FUNCTION_BLOCK RingToken (* Basic Function Block Type *)
  (* Standard: 61499-2 *)
  (* Version 0.2, 2003-12-04, JHC, Rockwell Automation, Renamed for better indexing. *)
  (* Version 0.1, 2002-11-05, JHC, Rockwell Automation, Corrected missing ST element in Algorithm REQ. *)
  (* Version 0.0, 2000-05-30, JHC, Rockwell Automation *)
  (* Compiler header: package fb.rt.cs725; *)
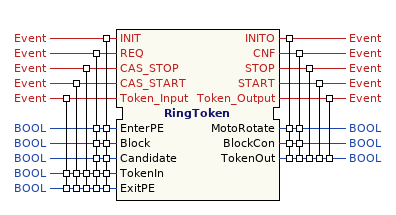
  EVENT_INPUT
    INIT WITH EnterPE, Block, Candidate, TokenIn, ExitPE; (* Initialization Request *)
    REQ WITH EnterPE, Block, Candidate, TokenIn, ExitPE; (* Normal Execution Request *)
    CAS_STOP WITH TokenIn, ExitPE;
    CAS_START WITH TokenIn, ExitPE;
    Token_Input WITH TokenIn, ExitPE;
  END_EVENT
  EVENT_OUTPUT
    INITO WITH MotoRotate, BlockCon, TokenOut; (* Initialization Confirm *)
    CNF WITH MotoRotate, BlockCon, TokenOut; (* Execution Confirmation *)
    STOP WITH TokenOut;
    START WITH TokenOut;
    Token_Output WITH TokenOut;
  END_EVENT
  VAR_INPUT
    EnterPE : BOOL; (* Input event qualifier *)
    Block : BOOL;
    Candidate : BOOL;
    TokenIn : BOOL;
    ExitPE : BOOL;
  END_VAR
  VAR_OUTPUT
    MotoRotate : BOOL; (* Output event qualifier *)
    BlockCon : BOOL;
    TokenOut : BOOL;
  END_VAR
  VAR
    lastPE : BOOL := 1;
    lastBlock : BOOL := 0;
  END_VAR
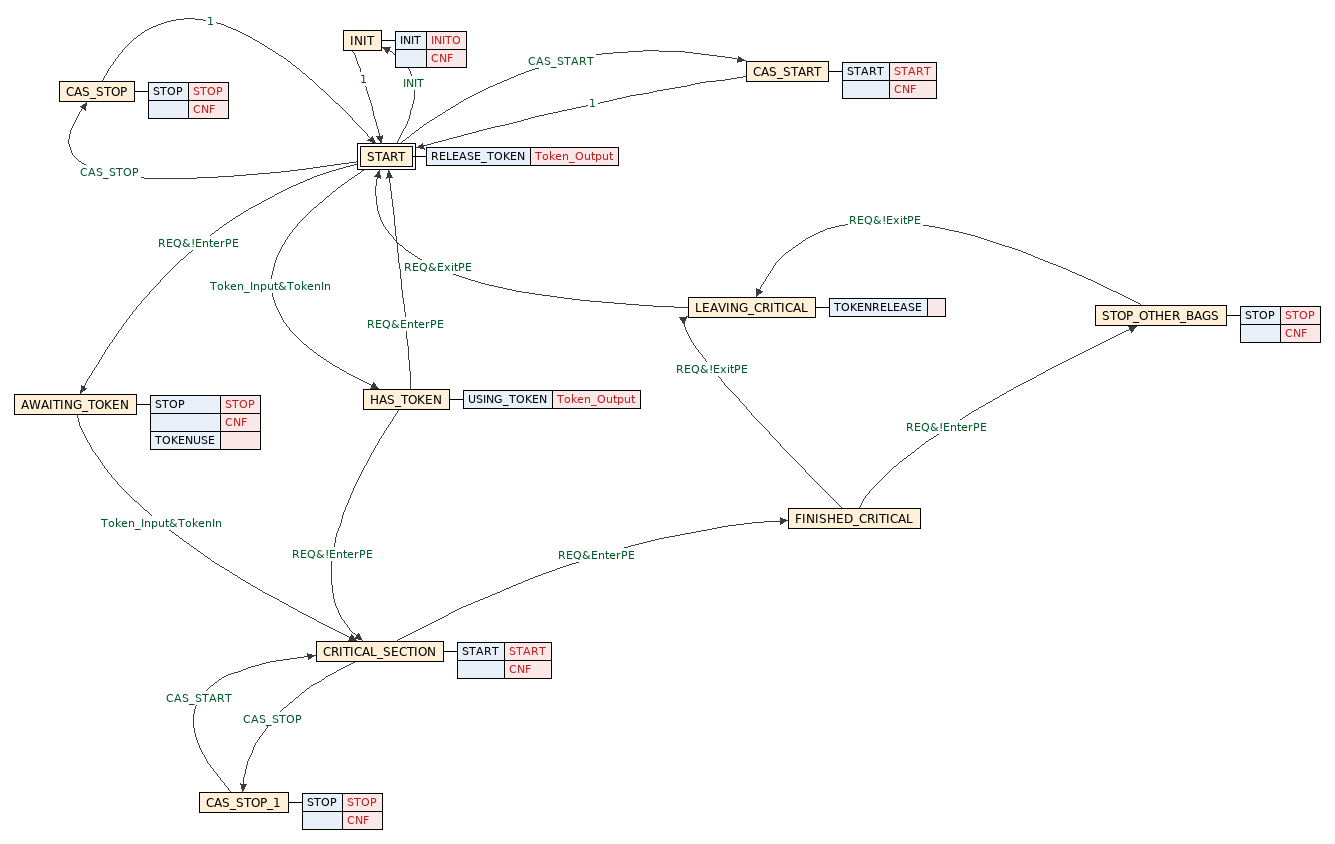
  EC_STATES
    START : RELEASE_TOKEN -> Token_Output;
    INIT : INIT -> INITO, -> CNF; (* Initialization *)
    AWAITING_TOKEN : STOP -> STOP, -> CNF, TOKENUSE; (* Waiting for token *)
    HAS_TOKEN : USING_TOKEN -> Token_Output;
    CRITICAL_SECTION : START -> START, -> CNF;
    FINISHED_CRITICAL;
    STOP_OTHER_BAGS : STOP -> STOP, -> CNF; (* Stop other incoming bags on the same conveyer *)
    LEAVING_CRITICAL : TOKENRELEASE;
    CAS_STOP : STOP -> STOP, -> CNF;
    CAS_START : START -> START, -> CNF;
    CAS_STOP_1 : STOP -> STOP, -> CNF;
  END_STATES
  EC_TRANSITIONS
    INIT TO START := 1;
    START TO AWAITING_TOKEN := REQ&!EnterPE;
    AWAITING_TOKEN TO CRITICAL_SECTION := Token_Input&TokenIn;
    HAS_TOKEN TO CRITICAL_SECTION := REQ&!EnterPE;
    START TO HAS_TOKEN := Token_Input&TokenIn;
    HAS_TOKEN TO START := REQ&EnterPE;
    CRITICAL_SECTION TO FINISHED_CRITICAL := REQ&EnterPE;
    START TO INIT := INIT;
    FINISHED_CRITICAL TO STOP_OTHER_BAGS := REQ&!EnterPE;
    FINISHED_CRITICAL TO LEAVING_CRITICAL := REQ&!ExitPE;
    STOP_OTHER_BAGS TO LEAVING_CRITICAL := REQ&!ExitPE;
    LEAVING_CRITICAL TO START := REQ&ExitPE;
    START TO CAS_STOP := CAS_STOP;
    CAS_STOP TO START := 1;
    START TO CAS_START := CAS_START;
    CAS_START TO START := 1;
    CRITICAL_SECTION TO CAS_STOP_1 := CAS_STOP;
    CAS_STOP_1 TO CRITICAL_SECTION := CAS_START;
  END_TRANSITIONS
  ALGORITHM INIT IN ST: (* Initialization algorithm *)
MotoRotate := TRUE;
Block := FALSE;
  END_ALGORITHM
  ALGORITHM REQ IN ST: (* Normally executed algorithm *)
IF Candidate THEN
IF lastPE !:= EnterPE THEN
IF NOT EnterPE THEN
BlockCon:= TRUE;
System.out.println("BlockCon = true");
ELSE
BlockCon:=FALSE;
System.out.println("BlockCon = false");
END_IF
lastPE := EnterPE;
END_IF
IF lastBlock !:= Block THEN
IF Block THEN
STOP.serviceEvent(this);
MotoRotate := FALSE;
System.out.println("Cas Stop");
ELSE
START.serviceEvent(this);
MotoRotate := TRUE;
System.out.println("Cas Start");
END_IF
lastBlock := Block;
END_IF
END_IF
  END_ALGORITHM
  ALGORITHM START IN ST:
MotoRotate:=TRUE;
  END_ALGORITHM
  ALGORITHM STOP IN ST:
MotoRotate := FALSE;
  END_ALGORITHM
  ALGORITHM USING_TOKEN IN ST:
TokenOut := FALSE;
  END_ALGORITHM
  ALGORITHM RELEASE_TOKEN IN ST:
TokenOut := TRUE;
  END_ALGORITHM
  ALGORITHM TOKENUSE IN ST:
System.out.println("Ring Token is being used");
  END_ALGORITHM
  ALGORITHM TOKENRELEASE IN ST:
System.out.println("Ring Token has been released");
  END_ALGORITHM
END_FUNCTION_BLOCK
